TYPE ST_Parent :
STRUCT
	stInner		: DUT_ServoRecipe;
	iMember		: DINT;
END_STRUCT
END_TYPE

(* stored: Version 1.1.0.1, ProductVersion 3.1.4024.12
   DUT ST_Parent: Id {4eda03c3-83f5-4e56-8ea8-292c743c20ed} *)
